TYPE "OOAx_Wng"
VERSION : 0.1
// Block: OOAx_Wng
   STRUCT
      SwLimitMinus : Bool;
      SwLimitPlus : Bool;
   END_STRUCT;

END_TYPE
